FUNCTION_BLOCK FB_LamparaConmutada_IL
// La lampara se enciende si estando apagada se acciona el pulsador
// La lampara se apaga si estando encendida se acciona el pulsador
VAR
    Pulsacion         : R_TRIG;
    Lampara   AT %Q*  : BOOL;
    Pulsador  AT %I*  : BOOL;
END_VAR

// NETWORK 1
// instruction list
CAL     Pulsacion(
    CLK     := Pulsador)

// NETWORK 2
// instruction list
LD      Pulsacion.Q
JMPCN   End

// NETWORK 3
// instruction list
LDN     Lampara
ST      Lampara

// NETWORK 4
End:
// instruction list

END_FUNCTION_BLOCK

(* stored: Version 1.1.0.1, ProductVersion 3.1.4024.15
   POU FB_LamparaConmutada_IL: Id {d1f54643-18b5-49e5-aa32-f8470987967d}, SpecialFunc None *)
